// TIA Portal V17 export
// export: Created 2025-06-26T06:49:19.2186578Z, ExportSetting WithDefaults, DisplayName Totally Integrated Automation Portal, DisplayVersion V17 Update 8, DisplayName TIA Portal Openness, DisplayVersion V17 Update 8, DisplayName TIA Portal Version Control Interface, DisplayVersion V17, DisplayName STEP 7 Professional, DisplayVersion V17 Update 8, DisplayName STEP 7 Safety, DisplayVersion V17 Update 6, DisplayName WinCC Advanced, DisplayVersion V17 Update 8
FUNCTION "WinCCAlarmHandling" : Void   // FC24, FBD
TITLE = Convert alarms to WinCC format
{ S7_Optimized_Access := 'TRUE' }
VERSION : 0.1
// stored: AutoNumber true, IsIECCheckEnabled false, SetENOAutomatically false, UDAEnableTagReadback false
BEGIN

REGION Network 1 (SCL): Comments
   (*
   For every alarm that should appear in the HMI, it has to be translated into WinCC's alarm format
   This is a very "dumb" way to do it, but the advantage is it's easy to understand and easy to modify.

   Steps to add a new alarm:
   1. Add an entry in DB_WinCCAlarms under the right category
   2. Add a network in this FC with a WinCCAlarm block
   3. In the WinCC project, import the tag from DB_WinCCAlarms
   4. In the WinCC project, create an alarm which references this tag
   *)
END_REGION

REGION Network 2: 0001
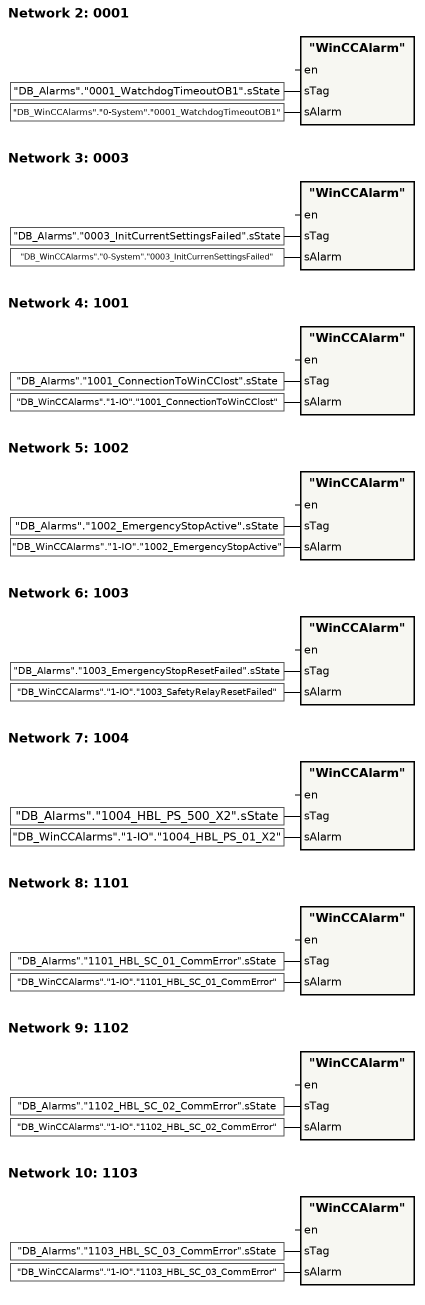
   "WinCCAlarm"(sTag := "DB_Alarms"."0001_WatchdogTimeoutOB1".sState,
                sAlarm := "DB_WinCCAlarms"."0-System"."0001_WatchdogTimeoutOB1");
END_REGION

REGION Network 3: 0003
   "WinCCAlarm"(sTag := "DB_Alarms"."0003_InitCurrentSettingsFailed".sState,
                sAlarm := "DB_WinCCAlarms"."0-System"."0003_InitCurrenSettingsFailed");
END_REGION

REGION Network 4: 1001
   "WinCCAlarm"(sTag := "DB_Alarms"."1001_ConnectionToWinCClost".sState,
                sAlarm := "DB_WinCCAlarms"."1-IO"."1001_ConnectionToWinCClost");
END_REGION

REGION Network 5: 1002
   "WinCCAlarm"(sTag := "DB_Alarms"."1002_EmergencyStopActive".sState,
                sAlarm := "DB_WinCCAlarms"."1-IO"."1002_EmergencyStopActive");
END_REGION

REGION Network 6: 1003
   "WinCCAlarm"(sTag := "DB_Alarms"."1003_EmergencyStopResetFailed".sState,
                sAlarm := "DB_WinCCAlarms"."1-IO"."1003_SafetyRelayResetFailed");
END_REGION

REGION Network 7: 1004
   "WinCCAlarm"(sTag := "DB_Alarms"."1004_HBL_PS_500_X2".sState,
                sAlarm := "DB_WinCCAlarms"."1-IO"."1004_HBL_PS_01_X2");
END_REGION

REGION Network 8: 1101
   "WinCCAlarm"(sTag := "DB_Alarms"."1101_HBL_SC_01_CommError".sState,
                sAlarm := "DB_WinCCAlarms"."1-IO"."1101_HBL_SC_01_CommError");
END_REGION

REGION Network 9: 1102
   "WinCCAlarm"(sTag := "DB_Alarms"."1102_HBL_SC_02_CommError".sState,
                sAlarm := "DB_WinCCAlarms"."1-IO"."1102_HBL_SC_02_CommError");
END_REGION

REGION Network 10: 1103
   "WinCCAlarm"(sTag := "DB_Alarms"."1103_HBL_SC_03_CommError".sState,
                sAlarm := "DB_WinCCAlarms"."1-IO"."1103_HBL_SC_03_CommError");
END_REGION

REGION Network 11: 1110
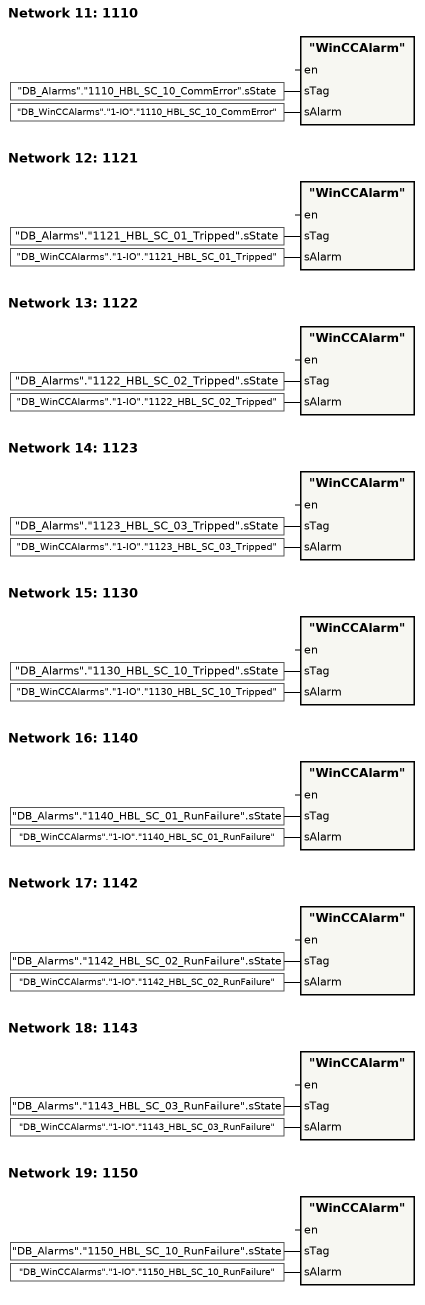
   "WinCCAlarm"(sTag := "DB_Alarms"."1110_HBL_SC_10_CommError".sState,
                sAlarm := "DB_WinCCAlarms"."1-IO"."1110_HBL_SC_10_CommError");
END_REGION

REGION Network 12: 1121
   "WinCCAlarm"(sTag := "DB_Alarms"."1121_HBL_SC_01_Tripped".sState,
                sAlarm := "DB_WinCCAlarms"."1-IO"."1121_HBL_SC_01_Tripped");
END_REGION

REGION Network 13: 1122
   "WinCCAlarm"(sTag := "DB_Alarms"."1122_HBL_SC_02_Tripped".sState,
                sAlarm := "DB_WinCCAlarms"."1-IO"."1122_HBL_SC_02_Tripped");
END_REGION

REGION Network 14: 1123
   "WinCCAlarm"(sTag := "DB_Alarms"."1123_HBL_SC_03_Tripped".sState,
                sAlarm := "DB_WinCCAlarms"."1-IO"."1123_HBL_SC_03_Tripped");
END_REGION

REGION Network 15: 1130
   "WinCCAlarm"(sTag := "DB_Alarms"."1130_HBL_SC_10_Tripped".sState,
                sAlarm := "DB_WinCCAlarms"."1-IO"."1130_HBL_SC_10_Tripped");
END_REGION

REGION Network 16: 1140
   "WinCCAlarm"(sTag := "DB_Alarms"."1140_HBL_SC_01_RunFailure".sState,
                sAlarm := "DB_WinCCAlarms"."1-IO"."1140_HBL_SC_01_RunFailure");
END_REGION

REGION Network 17: 1142
   "WinCCAlarm"(sTag := "DB_Alarms"."1142_HBL_SC_02_RunFailure".sState,
                sAlarm := "DB_WinCCAlarms"."1-IO"."1142_HBL_SC_02_RunFailure");
END_REGION

REGION Network 18: 1143
   "WinCCAlarm"(sTag := "DB_Alarms"."1143_HBL_SC_03_RunFailure".sState,
                sAlarm := "DB_WinCCAlarms"."1-IO"."1143_HBL_SC_03_RunFailure");
END_REGION

REGION Network 19: 1150
   "WinCCAlarm"(sTag := "DB_Alarms"."1150_HBL_SC_10_RunFailure".sState,
                sAlarm := "DB_WinCCAlarms"."1-IO"."1150_HBL_SC_10_RunFailure");
END_REGION

REGION Network 20: 1201
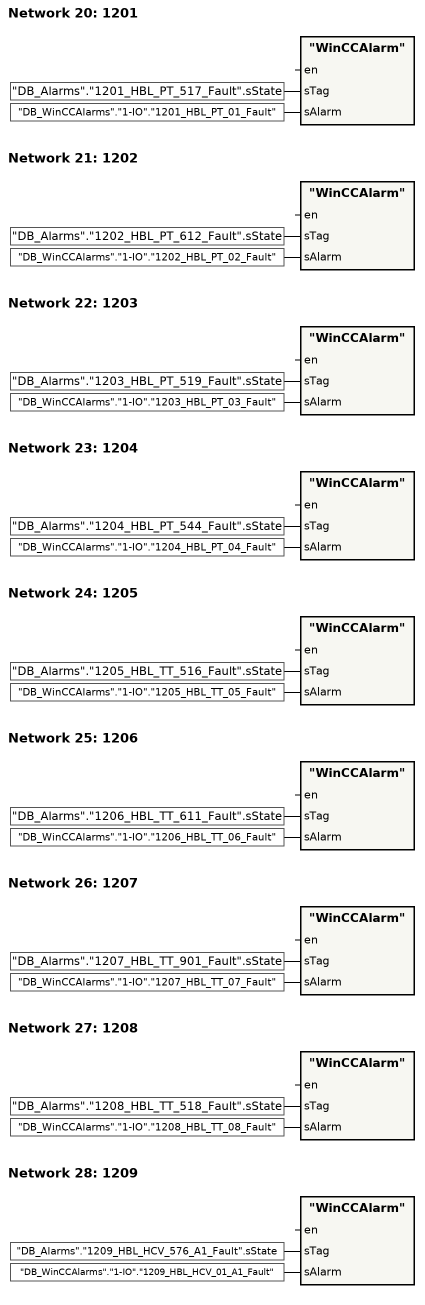
   "WinCCAlarm"(sTag := "DB_Alarms"."1201_HBL_PT_517_Fault".sState,
                sAlarm := "DB_WinCCAlarms"."1-IO"."1201_HBL_PT_01_Fault");
END_REGION

REGION Network 21: 1202
   "WinCCAlarm"(sTag := "DB_Alarms"."1202_HBL_PT_612_Fault".sState,
                sAlarm := "DB_WinCCAlarms"."1-IO"."1202_HBL_PT_02_Fault");
END_REGION

REGION Network 22: 1203
   "WinCCAlarm"(sTag := "DB_Alarms"."1203_HBL_PT_519_Fault".sState,
                sAlarm := "DB_WinCCAlarms"."1-IO"."1203_HBL_PT_03_Fault");
END_REGION

REGION Network 23: 1204
   "WinCCAlarm"(sTag := "DB_Alarms"."1204_HBL_PT_544_Fault".sState,
                sAlarm := "DB_WinCCAlarms"."1-IO"."1204_HBL_PT_04_Fault");
END_REGION

REGION Network 24: 1205
   "WinCCAlarm"(sTag := "DB_Alarms"."1205_HBL_TT_516_Fault".sState,
                sAlarm := "DB_WinCCAlarms"."1-IO"."1205_HBL_TT_05_Fault");
END_REGION

REGION Network 25: 1206
   "WinCCAlarm"(sTag := "DB_Alarms"."1206_HBL_TT_611_Fault".sState,
                sAlarm := "DB_WinCCAlarms"."1-IO"."1206_HBL_TT_06_Fault");
END_REGION

REGION Network 26: 1207
   "WinCCAlarm"(sTag := "DB_Alarms"."1207_HBL_TT_901_Fault".sState,
                sAlarm := "DB_WinCCAlarms"."1-IO"."1207_HBL_TT_07_Fault");
END_REGION

REGION Network 27: 1208
   "WinCCAlarm"(sTag := "DB_Alarms"."1208_HBL_TT_518_Fault".sState,
                sAlarm := "DB_WinCCAlarms"."1-IO"."1208_HBL_TT_08_Fault");
END_REGION

REGION Network 28: 1209
   "WinCCAlarm"(sTag := "DB_Alarms"."1209_HBL_HCV_576_A1_Fault".sState,
                sAlarm := "DB_WinCCAlarms"."1-IO"."1209_HBL_HCV_01_A1_Fault");
END_REGION

REGION Network 29: 1210
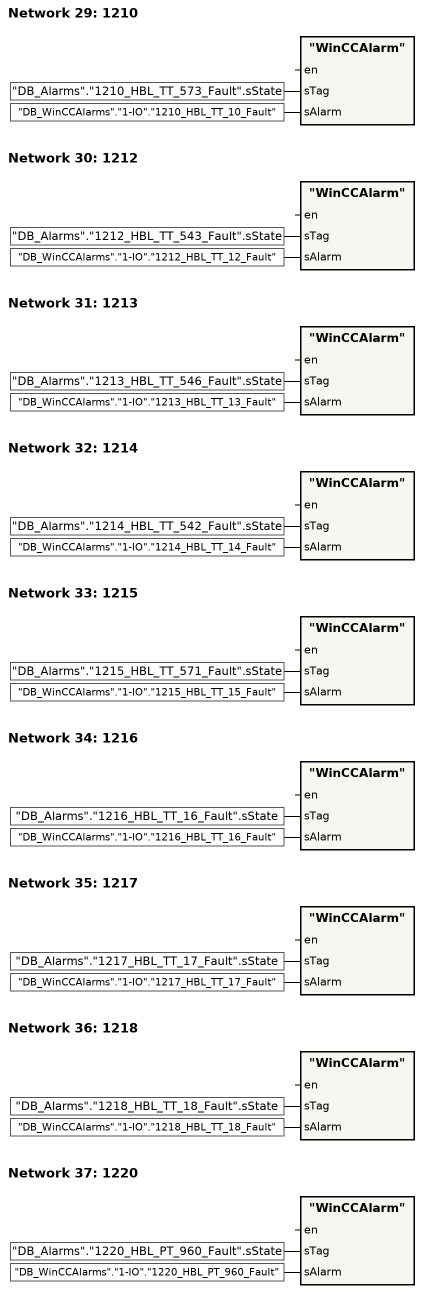
   "WinCCAlarm"(sTag := "DB_Alarms"."1210_HBL_TT_573_Fault".sState,
                sAlarm := "DB_WinCCAlarms"."1-IO"."1210_HBL_TT_10_Fault");
END_REGION

REGION Network 30: 1212
   "WinCCAlarm"(sTag := "DB_Alarms"."1212_HBL_TT_543_Fault".sState,
                sAlarm := "DB_WinCCAlarms"."1-IO"."1212_HBL_TT_12_Fault");
END_REGION

REGION Network 31: 1213
   "WinCCAlarm"(sTag := "DB_Alarms"."1213_HBL_TT_546_Fault".sState,
                sAlarm := "DB_WinCCAlarms"."1-IO"."1213_HBL_TT_13_Fault");
END_REGION

REGION Network 32: 1214
   "WinCCAlarm"(sTag := "DB_Alarms"."1214_HBL_TT_542_Fault".sState,
                sAlarm := "DB_WinCCAlarms"."1-IO"."1214_HBL_TT_14_Fault");
END_REGION

REGION Network 33: 1215
   "WinCCAlarm"(sTag := "DB_Alarms"."1215_HBL_TT_571_Fault".sState,
                sAlarm := "DB_WinCCAlarms"."1-IO"."1215_HBL_TT_15_Fault");
END_REGION

REGION Network 34: 1216
   "WinCCAlarm"(sTag := "DB_Alarms"."1216_HBL_TT_16_Fault".sState,
                sAlarm := "DB_WinCCAlarms"."1-IO"."1216_HBL_TT_16_Fault");
END_REGION

REGION Network 35: 1217
   "WinCCAlarm"(sTag := "DB_Alarms"."1217_HBL_TT_17_Fault".sState,
                sAlarm := "DB_WinCCAlarms"."1-IO"."1217_HBL_TT_17_Fault");
END_REGION

REGION Network 36: 1218
   "WinCCAlarm"(sTag := "DB_Alarms"."1218_HBL_TT_18_Fault".sState,
                sAlarm := "DB_WinCCAlarms"."1-IO"."1218_HBL_TT_18_Fault");
END_REGION

REGION Network 37: 1220
   "WinCCAlarm"(sTag := "DB_Alarms"."1220_HBL_PT_960_Fault".sState,
                sAlarm := "DB_WinCCAlarms"."1-IO"."1220_HBL_PT_960_Fault");
END_REGION

REGION Network 38: 1221
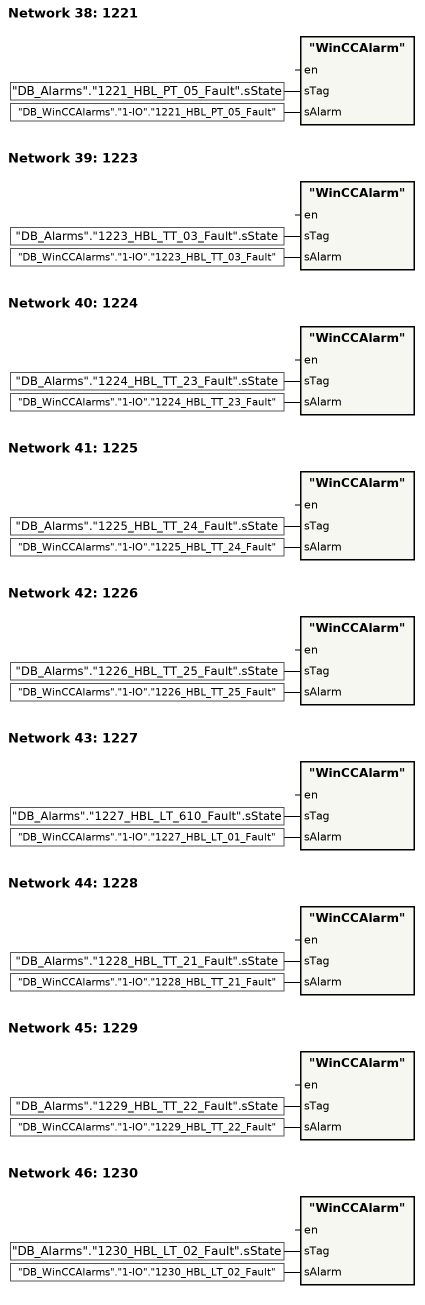
   "WinCCAlarm"(sTag := "DB_Alarms"."1221_HBL_PT_05_Fault".sState,
                sAlarm := "DB_WinCCAlarms"."1-IO"."1221_HBL_PT_05_Fault");
END_REGION

REGION Network 39: 1223
   "WinCCAlarm"(sTag := "DB_Alarms"."1223_HBL_TT_03_Fault".sState,
                sAlarm := "DB_WinCCAlarms"."1-IO"."1223_HBL_TT_03_Fault");
END_REGION

REGION Network 40: 1224
   "WinCCAlarm"(sTag := "DB_Alarms"."1224_HBL_TT_23_Fault".sState,
                sAlarm := "DB_WinCCAlarms"."1-IO"."1224_HBL_TT_23_Fault");
END_REGION

REGION Network 41: 1225
   "WinCCAlarm"(sTag := "DB_Alarms"."1225_HBL_TT_24_Fault".sState,
                sAlarm := "DB_WinCCAlarms"."1-IO"."1225_HBL_TT_24_Fault");
END_REGION

REGION Network 42: 1226
   "WinCCAlarm"(sTag := "DB_Alarms"."1226_HBL_TT_25_Fault".sState,
                sAlarm := "DB_WinCCAlarms"."1-IO"."1226_HBL_TT_25_Fault");
END_REGION

REGION Network 43: 1227
   "WinCCAlarm"(sTag := "DB_Alarms"."1227_HBL_LT_610_Fault".sState,
                sAlarm := "DB_WinCCAlarms"."1-IO"."1227_HBL_LT_01_Fault");
END_REGION

REGION Network 44: 1228
   "WinCCAlarm"(sTag := "DB_Alarms"."1228_HBL_TT_21_Fault".sState,
                sAlarm := "DB_WinCCAlarms"."1-IO"."1228_HBL_TT_21_Fault");
END_REGION

REGION Network 45: 1229
   "WinCCAlarm"(sTag := "DB_Alarms"."1229_HBL_TT_22_Fault".sState,
                sAlarm := "DB_WinCCAlarms"."1-IO"."1229_HBL_TT_22_Fault");
END_REGION

REGION Network 46: 1230
   "WinCCAlarm"(sTag := "DB_Alarms"."1230_HBL_LT_02_Fault".sState,
                sAlarm := "DB_WinCCAlarms"."1-IO"."1230_HBL_LT_02_Fault");
END_REGION

REGION Network 47: 1231
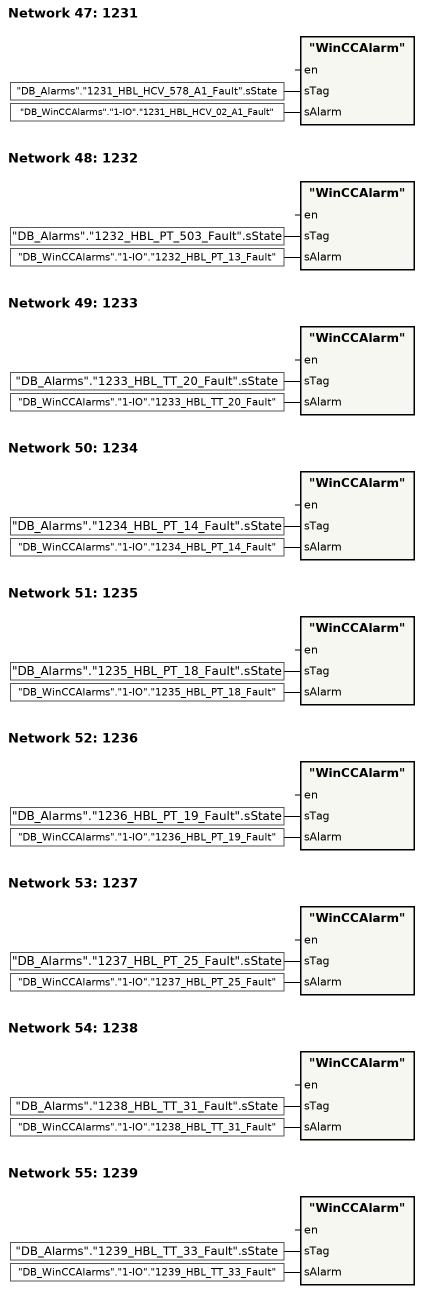
   "WinCCAlarm"(sTag := "DB_Alarms"."1231_HBL_HCV_578_A1_Fault".sState,
                sAlarm := "DB_WinCCAlarms"."1-IO"."1231_HBL_HCV_02_A1_Fault");
END_REGION

REGION Network 48: 1232
   "WinCCAlarm"(sTag := "DB_Alarms"."1232_HBL_PT_503_Fault".sState,
                sAlarm := "DB_WinCCAlarms"."1-IO"."1232_HBL_PT_13_Fault");
END_REGION

REGION Network 49: 1233
   "WinCCAlarm"(sTag := "DB_Alarms"."1233_HBL_TT_20_Fault".sState,
                sAlarm := "DB_WinCCAlarms"."1-IO"."1233_HBL_TT_20_Fault");
END_REGION

REGION Network 50: 1234
   "WinCCAlarm"(sTag := "DB_Alarms"."1234_HBL_PT_14_Fault".sState,
                sAlarm := "DB_WinCCAlarms"."1-IO"."1234_HBL_PT_14_Fault");
END_REGION

REGION Network 51: 1235
   "WinCCAlarm"(sTag := "DB_Alarms"."1235_HBL_PT_18_Fault".sState,
                sAlarm := "DB_WinCCAlarms"."1-IO"."1235_HBL_PT_18_Fault");
END_REGION

REGION Network 52: 1236
   "WinCCAlarm"(sTag := "DB_Alarms"."1236_HBL_PT_19_Fault".sState,
                sAlarm := "DB_WinCCAlarms"."1-IO"."1236_HBL_PT_19_Fault");
END_REGION

REGION Network 53: 1237
   "WinCCAlarm"(sTag := "DB_Alarms"."1237_HBL_PT_25_Fault".sState,
                sAlarm := "DB_WinCCAlarms"."1-IO"."1237_HBL_PT_25_Fault");
END_REGION

REGION Network 54: 1238
   "WinCCAlarm"(sTag := "DB_Alarms"."1238_HBL_TT_31_Fault".sState,
                sAlarm := "DB_WinCCAlarms"."1-IO"."1238_HBL_TT_31_Fault");
END_REGION

REGION Network 55: 1239
   "WinCCAlarm"(sTag := "DB_Alarms"."1239_HBL_TT_33_Fault".sState,
                sAlarm := "DB_WinCCAlarms"."1-IO"."1239_HBL_TT_33_Fault");
END_REGION

REGION Network 56: 1240
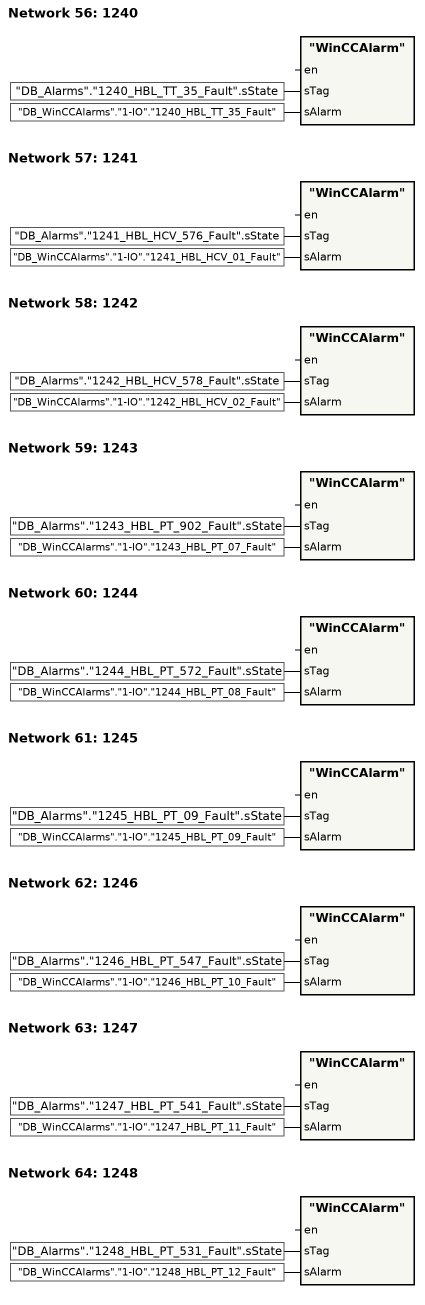
   "WinCCAlarm"(sTag := "DB_Alarms"."1240_HBL_TT_35_Fault".sState,
                sAlarm := "DB_WinCCAlarms"."1-IO"."1240_HBL_TT_35_Fault");
END_REGION

REGION Network 57: 1241
   "WinCCAlarm"(sTag := "DB_Alarms"."1241_HBL_HCV_576_Fault".sState,
                sAlarm := "DB_WinCCAlarms"."1-IO"."1241_HBL_HCV_01_Fault");
END_REGION

REGION Network 58: 1242
   "WinCCAlarm"(sTag := "DB_Alarms"."1242_HBL_HCV_578_Fault".sState,
                sAlarm := "DB_WinCCAlarms"."1-IO"."1242_HBL_HCV_02_Fault");
END_REGION

REGION Network 59: 1243
   "WinCCAlarm"(sTag := "DB_Alarms"."1243_HBL_PT_902_Fault".sState,
                sAlarm := "DB_WinCCAlarms"."1-IO"."1243_HBL_PT_07_Fault");
END_REGION

REGION Network 60: 1244
   "WinCCAlarm"(sTag := "DB_Alarms"."1244_HBL_PT_572_Fault".sState,
                sAlarm := "DB_WinCCAlarms"."1-IO"."1244_HBL_PT_08_Fault");
END_REGION

REGION Network 61: 1245
   "WinCCAlarm"(sTag := "DB_Alarms"."1245_HBL_PT_09_Fault".sState,
                sAlarm := "DB_WinCCAlarms"."1-IO"."1245_HBL_PT_09_Fault");
END_REGION

REGION Network 62: 1246
   "WinCCAlarm"(sTag := "DB_Alarms"."1246_HBL_PT_547_Fault".sState,
                sAlarm := "DB_WinCCAlarms"."1-IO"."1246_HBL_PT_10_Fault");
END_REGION

REGION Network 63: 1247
   "WinCCAlarm"(sTag := "DB_Alarms"."1247_HBL_PT_541_Fault".sState,
                sAlarm := "DB_WinCCAlarms"."1-IO"."1247_HBL_PT_11_Fault");
END_REGION

REGION Network 64: 1248
   "WinCCAlarm"(sTag := "DB_Alarms"."1248_HBL_PT_531_Fault".sState,
                sAlarm := "DB_WinCCAlarms"."1-IO"."1248_HBL_PT_12_Fault");
END_REGION

REGION Network 65: 1249
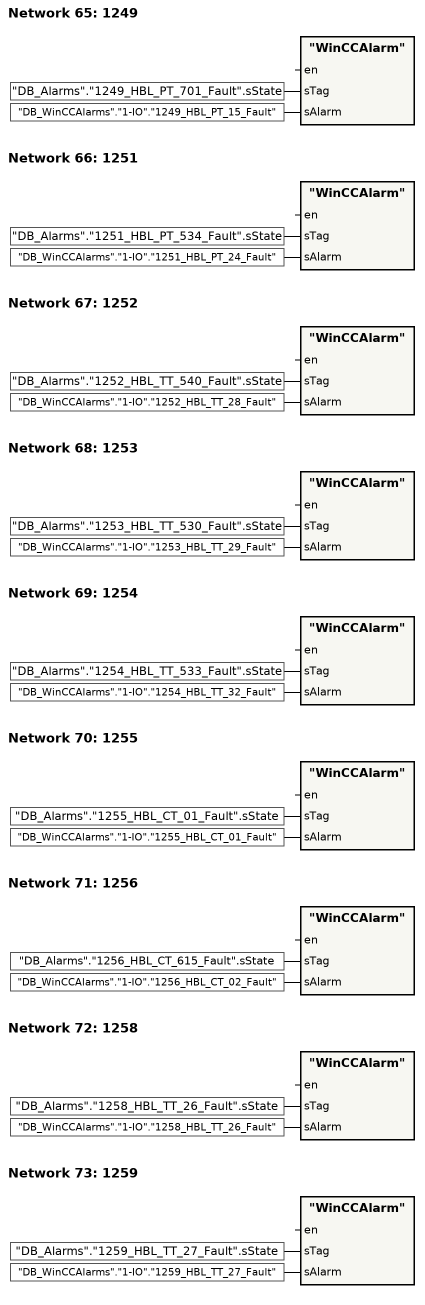
   "WinCCAlarm"(sTag := "DB_Alarms"."1249_HBL_PT_701_Fault".sState,
                sAlarm := "DB_WinCCAlarms"."1-IO"."1249_HBL_PT_15_Fault");
END_REGION

REGION Network 66: 1251
   "WinCCAlarm"(sTag := "DB_Alarms"."1251_HBL_PT_534_Fault".sState,
                sAlarm := "DB_WinCCAlarms"."1-IO"."1251_HBL_PT_24_Fault");
END_REGION

REGION Network 67: 1252
   "WinCCAlarm"(sTag := "DB_Alarms"."1252_HBL_TT_540_Fault".sState,
                sAlarm := "DB_WinCCAlarms"."1-IO"."1252_HBL_TT_28_Fault");
END_REGION

REGION Network 68: 1253
   "WinCCAlarm"(sTag := "DB_Alarms"."1253_HBL_TT_530_Fault".sState,
                sAlarm := "DB_WinCCAlarms"."1-IO"."1253_HBL_TT_29_Fault");
END_REGION

REGION Network 69: 1254
   "WinCCAlarm"(sTag := "DB_Alarms"."1254_HBL_TT_533_Fault".sState,
                sAlarm := "DB_WinCCAlarms"."1-IO"."1254_HBL_TT_32_Fault");
END_REGION

REGION Network 70: 1255
   "WinCCAlarm"(sTag := "DB_Alarms"."1255_HBL_CT_01_Fault".sState,
                sAlarm := "DB_WinCCAlarms"."1-IO"."1255_HBL_CT_01_Fault");
END_REGION

REGION Network 71: 1256
   "WinCCAlarm"(sTag := "DB_Alarms"."1256_HBL_CT_615_Fault".sState,
                sAlarm := "DB_WinCCAlarms"."1-IO"."1256_HBL_CT_02_Fault");
END_REGION

REGION Network 72: 1258
   "WinCCAlarm"(sTag := "DB_Alarms"."1258_HBL_TT_26_Fault".sState,
                sAlarm := "DB_WinCCAlarms"."1-IO"."1258_HBL_TT_26_Fault");
END_REGION

REGION Network 73: 1259
   "WinCCAlarm"(sTag := "DB_Alarms"."1259_HBL_TT_27_Fault".sState,
                sAlarm := "DB_WinCCAlarms"."1-IO"."1259_HBL_TT_27_Fault");
END_REGION

REGION Network 74: 1260
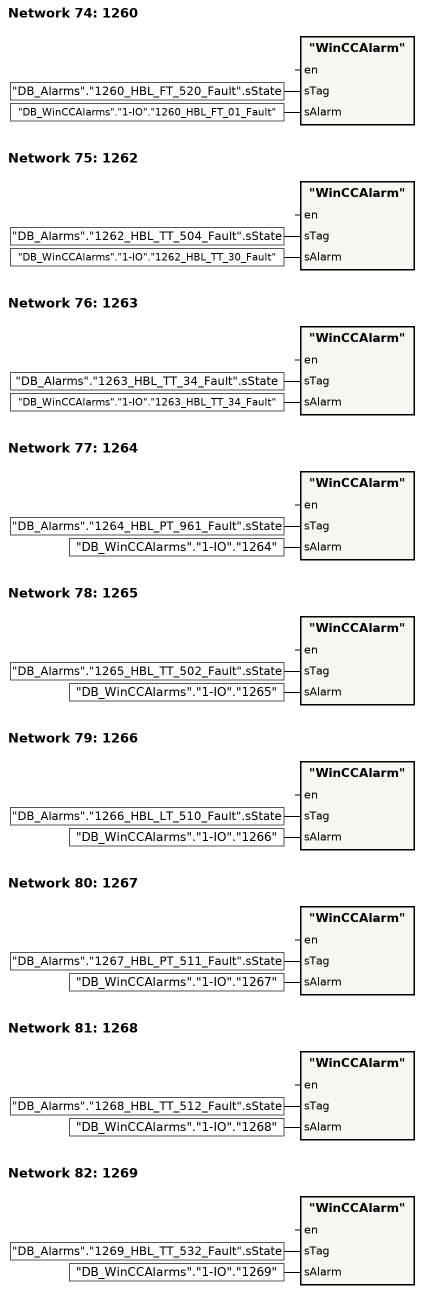
   "WinCCAlarm"(sTag := "DB_Alarms"."1260_HBL_FT_520_Fault".sState,
                sAlarm := "DB_WinCCAlarms"."1-IO"."1260_HBL_FT_01_Fault");
END_REGION

REGION Network 75: 1262
   "WinCCAlarm"(sTag := "DB_Alarms"."1262_HBL_TT_504_Fault".sState,
                sAlarm := "DB_WinCCAlarms"."1-IO"."1262_HBL_TT_30_Fault");
END_REGION

REGION Network 76: 1263
   "WinCCAlarm"(sTag := "DB_Alarms"."1263_HBL_TT_34_Fault".sState,
                sAlarm := "DB_WinCCAlarms"."1-IO"."1263_HBL_TT_34_Fault");
END_REGION

REGION Network 77: 1264
   "WinCCAlarm"(sTag := "DB_Alarms"."1264_HBL_PT_961_Fault".sState, sAlarm := "DB_WinCCAlarms"."1-IO"."1264");
END_REGION

REGION Network 78: 1265
   "WinCCAlarm"(sTag := "DB_Alarms"."1265_HBL_TT_502_Fault".sState, sAlarm := "DB_WinCCAlarms"."1-IO"."1265");
END_REGION

REGION Network 79: 1266
   "WinCCAlarm"(sTag := "DB_Alarms"."1266_HBL_LT_510_Fault".sState, sAlarm := "DB_WinCCAlarms"."1-IO"."1266");
END_REGION

REGION Network 80: 1267
   "WinCCAlarm"(sTag := "DB_Alarms"."1267_HBL_PT_511_Fault".sState, sAlarm := "DB_WinCCAlarms"."1-IO"."1267");
END_REGION

REGION Network 81: 1268
   "WinCCAlarm"(sTag := "DB_Alarms"."1268_HBL_TT_512_Fault".sState, sAlarm := "DB_WinCCAlarms"."1-IO"."1268");
END_REGION

REGION Network 82: 1269
   "WinCCAlarm"(sTag := "DB_Alarms"."1269_HBL_TT_532_Fault".sState, sAlarm := "DB_WinCCAlarms"."1-IO"."1269");
END_REGION

REGION Network 83: 1270
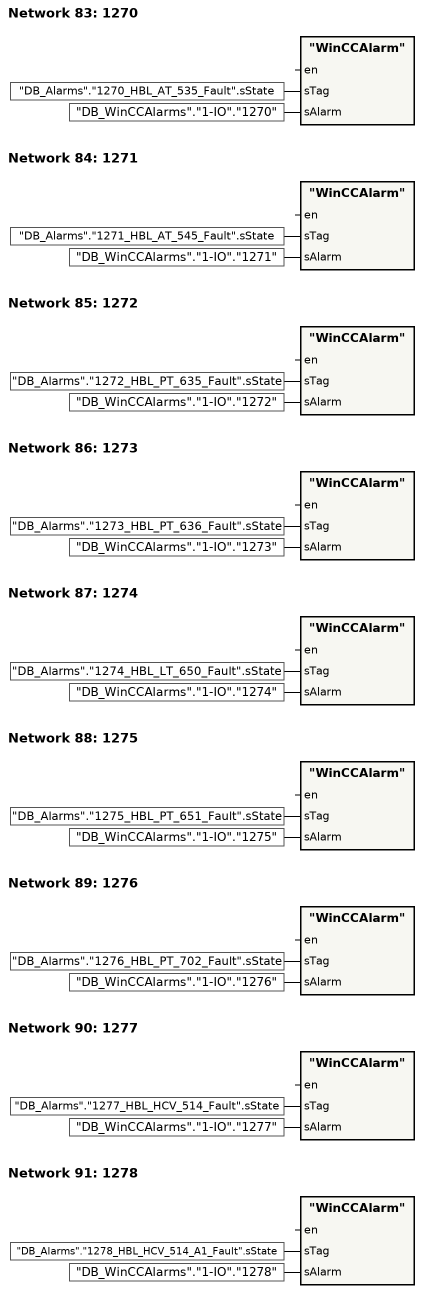
   "WinCCAlarm"(sTag := "DB_Alarms"."1270_HBL_AT_535_Fault".sState, sAlarm := "DB_WinCCAlarms"."1-IO"."1270");
END_REGION

REGION Network 84: 1271
   "WinCCAlarm"(sTag := "DB_Alarms"."1271_HBL_AT_545_Fault".sState, sAlarm := "DB_WinCCAlarms"."1-IO"."1271");
END_REGION

REGION Network 85: 1272
   "WinCCAlarm"(sTag := "DB_Alarms"."1272_HBL_PT_635_Fault".sState, sAlarm := "DB_WinCCAlarms"."1-IO"."1272");
END_REGION

REGION Network 86: 1273
   "WinCCAlarm"(sTag := "DB_Alarms"."1273_HBL_PT_636_Fault".sState, sAlarm := "DB_WinCCAlarms"."1-IO"."1273");
END_REGION

REGION Network 87: 1274
   "WinCCAlarm"(sTag := "DB_Alarms"."1274_HBL_LT_650_Fault".sState, sAlarm := "DB_WinCCAlarms"."1-IO"."1274");
END_REGION

REGION Network 88: 1275
   "WinCCAlarm"(sTag := "DB_Alarms"."1275_HBL_PT_651_Fault".sState, sAlarm := "DB_WinCCAlarms"."1-IO"."1275");
END_REGION

REGION Network 89: 1276
   "WinCCAlarm"(sTag := "DB_Alarms"."1276_HBL_PT_702_Fault".sState, sAlarm := "DB_WinCCAlarms"."1-IO"."1276");
END_REGION

REGION Network 90: 1277
   "WinCCAlarm"(sTag := "DB_Alarms"."1277_HBL_HCV_514_Fault".sState, sAlarm := "DB_WinCCAlarms"."1-IO"."1277");
END_REGION

REGION Network 91: 1278
   "WinCCAlarm"(sTag := "DB_Alarms"."1278_HBL_HCV_514_A1_Fault".sState,
                sAlarm := "DB_WinCCAlarms"."1-IO"."1278");
END_REGION

REGION Network 92: 1279
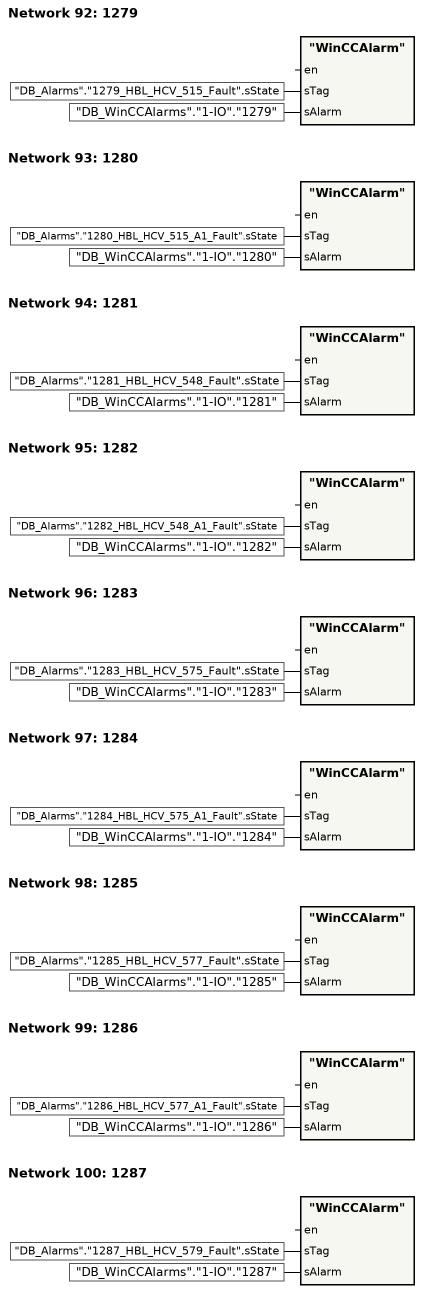
   "WinCCAlarm"(sTag := "DB_Alarms"."1279_HBL_HCV_515_Fault".sState, sAlarm := "DB_WinCCAlarms"."1-IO"."1279");
END_REGION

REGION Network 93: 1280
   "WinCCAlarm"(sTag := "DB_Alarms"."1280_HBL_HCV_515_A1_Fault".sState,
                sAlarm := "DB_WinCCAlarms"."1-IO"."1280");
END_REGION

REGION Network 94: 1281
   "WinCCAlarm"(sTag := "DB_Alarms"."1281_HBL_HCV_548_Fault".sState, sAlarm := "DB_WinCCAlarms"."1-IO"."1281");
END_REGION

REGION Network 95: 1282
   "WinCCAlarm"(sTag := "DB_Alarms"."1282_HBL_HCV_548_A1_Fault".sState,
                sAlarm := "DB_WinCCAlarms"."1-IO"."1282");
END_REGION

REGION Network 96: 1283
   "WinCCAlarm"(sTag := "DB_Alarms"."1283_HBL_HCV_575_Fault".sState, sAlarm := "DB_WinCCAlarms"."1-IO"."1283");
END_REGION

REGION Network 97: 1284
   "WinCCAlarm"(sTag := "DB_Alarms"."1284_HBL_HCV_575_A1_Fault".sState,
                sAlarm := "DB_WinCCAlarms"."1-IO"."1284");
END_REGION

REGION Network 98: 1285
   "WinCCAlarm"(sTag := "DB_Alarms"."1285_HBL_HCV_577_Fault".sState, sAlarm := "DB_WinCCAlarms"."1-IO"."1285");
END_REGION

REGION Network 99: 1286
   "WinCCAlarm"(sTag := "DB_Alarms"."1286_HBL_HCV_577_A1_Fault".sState,
                sAlarm := "DB_WinCCAlarms"."1-IO"."1286");
END_REGION

REGION Network 100: 1287
   "WinCCAlarm"(sTag := "DB_Alarms"."1287_HBL_HCV_579_Fault".sState, sAlarm := "DB_WinCCAlarms"."1-IO"."1287");
END_REGION

REGION Network 101: 1288
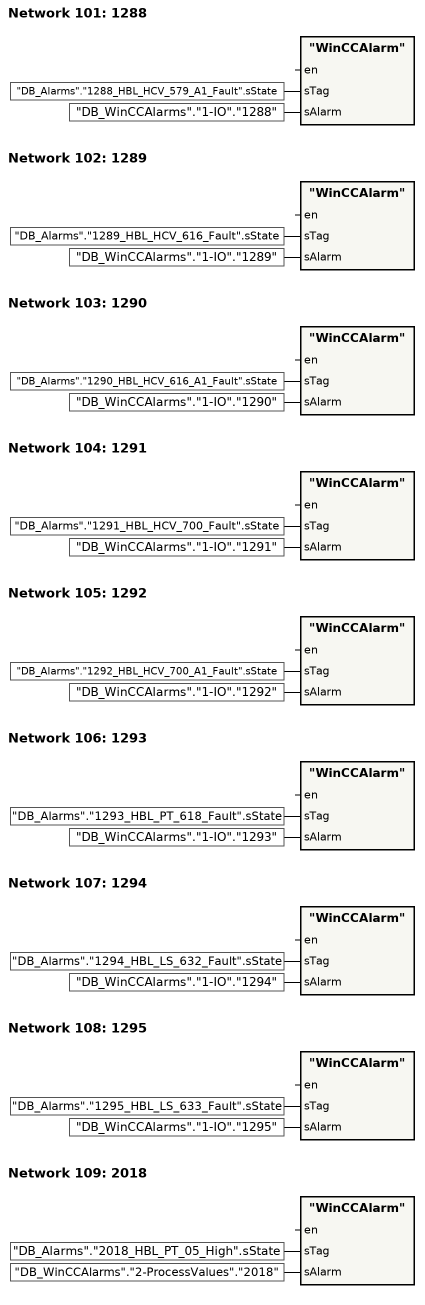
   "WinCCAlarm"(sTag := "DB_Alarms"."1288_HBL_HCV_579_A1_Fault".sState,
                sAlarm := "DB_WinCCAlarms"."1-IO"."1288");
END_REGION

REGION Network 102: 1289
   "WinCCAlarm"(sTag := "DB_Alarms"."1289_HBL_HCV_616_Fault".sState, sAlarm := "DB_WinCCAlarms"."1-IO"."1289");
END_REGION

REGION Network 103: 1290
   "WinCCAlarm"(sTag := "DB_Alarms"."1290_HBL_HCV_616_A1_Fault".sState,
                sAlarm := "DB_WinCCAlarms"."1-IO"."1290");
END_REGION

REGION Network 104: 1291
   "WinCCAlarm"(sTag := "DB_Alarms"."1291_HBL_HCV_700_Fault".sState, sAlarm := "DB_WinCCAlarms"."1-IO"."1291");
END_REGION

REGION Network 105: 1292
   "WinCCAlarm"(sTag := "DB_Alarms"."1292_HBL_HCV_700_A1_Fault".sState,
                sAlarm := "DB_WinCCAlarms"."1-IO"."1292");
END_REGION

REGION Network 106: 1293
   "WinCCAlarm"(sTag := "DB_Alarms"."1293_HBL_PT_618_Fault".sState, sAlarm := "DB_WinCCAlarms"."1-IO"."1293");
END_REGION

REGION Network 107: 1294
   "WinCCAlarm"(sTag := "DB_Alarms"."1294_HBL_LS_632_Fault".sState, sAlarm := "DB_WinCCAlarms"."1-IO"."1294");
END_REGION

REGION Network 108: 1295
   "WinCCAlarm"(sTag := "DB_Alarms"."1295_HBL_LS_633_Fault".sState, sAlarm := "DB_WinCCAlarms"."1-IO"."1295");
END_REGION

REGION Network 109: 2018
   "WinCCAlarm"(sTag := "DB_Alarms"."2018_HBL_PT_05_High".sState,
                sAlarm := "DB_WinCCAlarms"."2-ProcessValues"."2018");
END_REGION

REGION Network 110: 2028
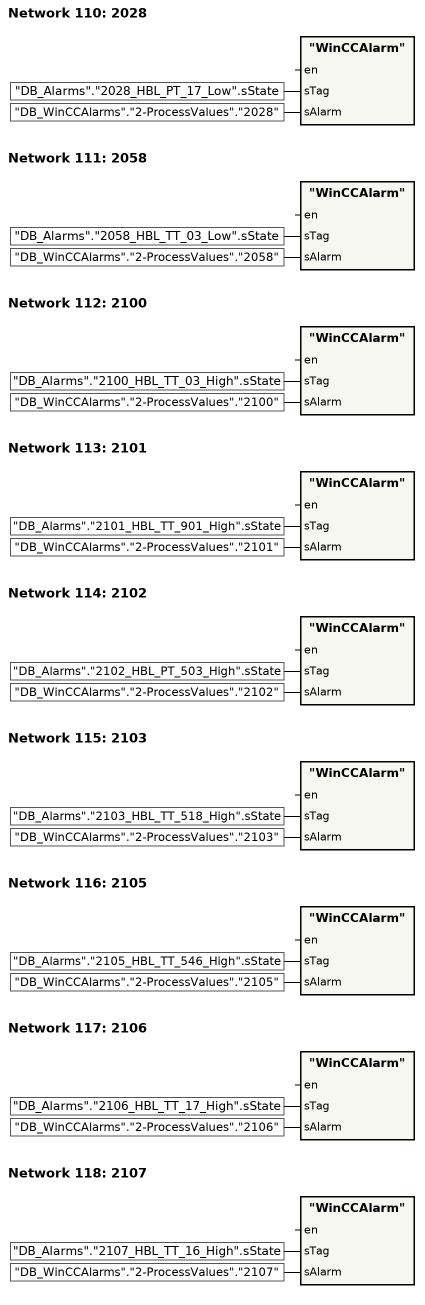
   "WinCCAlarm"(sTag := "DB_Alarms"."2028_HBL_PT_17_Low".sState,
                sAlarm := "DB_WinCCAlarms"."2-ProcessValues"."2028");
END_REGION

REGION Network 111: 2058
   "WinCCAlarm"(sTag := "DB_Alarms"."2058_HBL_TT_03_Low".sState,
                sAlarm := "DB_WinCCAlarms"."2-ProcessValues"."2058");
END_REGION

REGION Network 112: 2100
   "WinCCAlarm"(sTag := "DB_Alarms"."2100_HBL_TT_03_High".sState,
                sAlarm := "DB_WinCCAlarms"."2-ProcessValues"."2100");
END_REGION

REGION Network 113: 2101
   "WinCCAlarm"(sTag := "DB_Alarms"."2101_HBL_TT_901_High".sState,
                sAlarm := "DB_WinCCAlarms"."2-ProcessValues"."2101");
END_REGION

REGION Network 114: 2102
   "WinCCAlarm"(sTag := "DB_Alarms"."2102_HBL_PT_503_High".sState,
                sAlarm := "DB_WinCCAlarms"."2-ProcessValues"."2102");
END_REGION

REGION Network 115: 2103
   "WinCCAlarm"(sTag := "DB_Alarms"."2103_HBL_TT_518_High".sState,
                sAlarm := "DB_WinCCAlarms"."2-ProcessValues"."2103");
END_REGION

REGION Network 116: 2105
   "WinCCAlarm"(sTag := "DB_Alarms"."2105_HBL_TT_546_High".sState,
                sAlarm := "DB_WinCCAlarms"."2-ProcessValues"."2105");
END_REGION

REGION Network 117: 2106
   "WinCCAlarm"(sTag := "DB_Alarms"."2106_HBL_TT_17_High".sState,
                sAlarm := "DB_WinCCAlarms"."2-ProcessValues"."2106");
END_REGION

REGION Network 118: 2107
   "WinCCAlarm"(sTag := "DB_Alarms"."2107_HBL_TT_16_High".sState,
                sAlarm := "DB_WinCCAlarms"."2-ProcessValues"."2107");
END_REGION

REGION Network 119: 2108
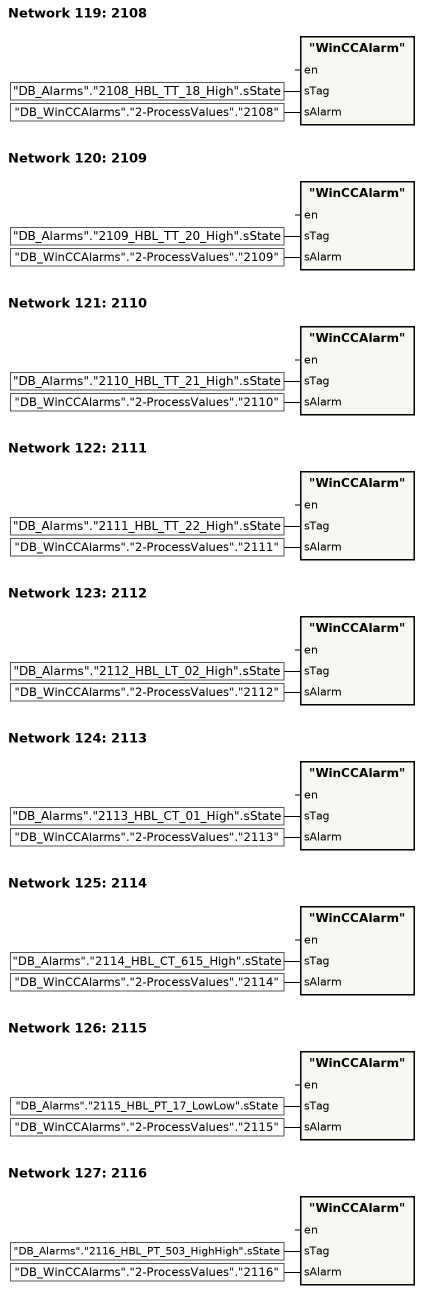
   "WinCCAlarm"(sTag := "DB_Alarms"."2108_HBL_TT_18_High".sState,
                sAlarm := "DB_WinCCAlarms"."2-ProcessValues"."2108");
END_REGION

REGION Network 120: 2109
   "WinCCAlarm"(sTag := "DB_Alarms"."2109_HBL_TT_20_High".sState,
                sAlarm := "DB_WinCCAlarms"."2-ProcessValues"."2109");
END_REGION

REGION Network 121: 2110
   "WinCCAlarm"(sTag := "DB_Alarms"."2110_HBL_TT_21_High".sState,
                sAlarm := "DB_WinCCAlarms"."2-ProcessValues"."2110");
END_REGION

REGION Network 122: 2111
   "WinCCAlarm"(sTag := "DB_Alarms"."2111_HBL_TT_22_High".sState,
                sAlarm := "DB_WinCCAlarms"."2-ProcessValues"."2111");
END_REGION

REGION Network 123: 2112
   "WinCCAlarm"(sTag := "DB_Alarms"."2112_HBL_LT_02_High".sState,
                sAlarm := "DB_WinCCAlarms"."2-ProcessValues"."2112");
END_REGION

REGION Network 124: 2113
   "WinCCAlarm"(sTag := "DB_Alarms"."2113_HBL_CT_01_High".sState,
                sAlarm := "DB_WinCCAlarms"."2-ProcessValues"."2113");
END_REGION

REGION Network 125: 2114
   "WinCCAlarm"(sTag := "DB_Alarms"."2114_HBL_CT_615_High".sState,
                sAlarm := "DB_WinCCAlarms"."2-ProcessValues"."2114");
END_REGION

REGION Network 126: 2115
   "WinCCAlarm"(sTag := "DB_Alarms"."2115_HBL_PT_17_LowLow".sState,
                sAlarm := "DB_WinCCAlarms"."2-ProcessValues"."2115");
END_REGION

REGION Network 127: 2116
   "WinCCAlarm"(sTag := "DB_Alarms"."2116_HBL_PT_503_HighHigh".sState,
                sAlarm := "DB_WinCCAlarms"."2-ProcessValues"."2116");
END_REGION

REGION Network 128: 2117
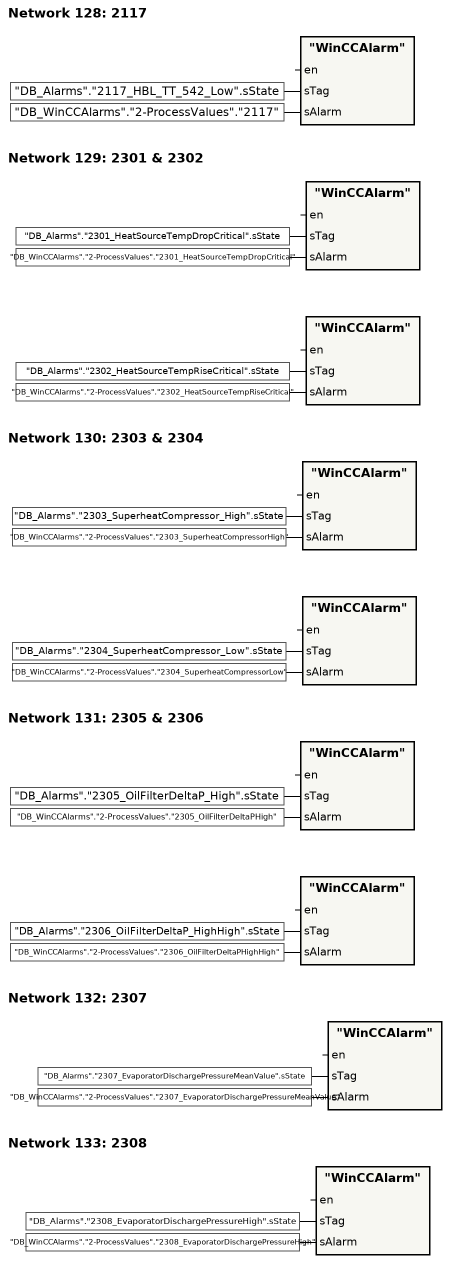
   "WinCCAlarm"(sTag := "DB_Alarms"."2117_HBL_TT_542_Low".sState,
                sAlarm := "DB_WinCCAlarms"."2-ProcessValues"."2117");
END_REGION

REGION Network 129: 2301 & 2302
   "WinCCAlarm"(sTag := "DB_Alarms"."2301_HeatSourceTempDropCritical".sState,
                sAlarm := "DB_WinCCAlarms"."2-ProcessValues"."2301_HeatSourceTempDropCritical");
   "WinCCAlarm"(sTag := "DB_Alarms"."2302_HeatSourceTempRiseCritical".sState,
                sAlarm := "DB_WinCCAlarms"."2-ProcessValues"."2302_HeatSourceTempRiseCritical");
END_REGION

REGION Network 130: 2303 & 2304
   "WinCCAlarm"(sTag := "DB_Alarms"."2303_SuperheatCompressor_High".sState,
                sAlarm := "DB_WinCCAlarms"."2-ProcessValues"."2303_SuperheatCompressorHigh");
   "WinCCAlarm"(sTag := "DB_Alarms"."2304_SuperheatCompressor_Low".sState,
                sAlarm := "DB_WinCCAlarms"."2-ProcessValues"."2304_SuperheatCompressorLow");
END_REGION

REGION Network 131: 2305 & 2306
   "WinCCAlarm"(sTag := "DB_Alarms"."2305_OilFilterDeltaP_High".sState,
                sAlarm := "DB_WinCCAlarms"."2-ProcessValues"."2305_OilFilterDeltaPHigh");
   "WinCCAlarm"(sTag := "DB_Alarms"."2306_OilFilterDeltaP_HighHigh".sState,
                sAlarm := "DB_WinCCAlarms"."2-ProcessValues"."2306_OilFilterDeltaPHighHigh");
END_REGION

REGION Network 132: 2307
   "WinCCAlarm"(sTag := "DB_Alarms"."2307_EvaporatorDischargePressureMeanValue".sState,
                sAlarm := "DB_WinCCAlarms"."2-ProcessValues"."2307_EvaporatorDischargePressureMeanValue");
END_REGION

REGION Network 133: 2308
   "WinCCAlarm"(sTag := "DB_Alarms"."2308_EvaporatorDischargePressureHigh".sState,
                sAlarm := "DB_WinCCAlarms"."2-ProcessValues"."2308_EvaporatorDischargePressureHigh");
END_REGION

REGION Network 134: 2309
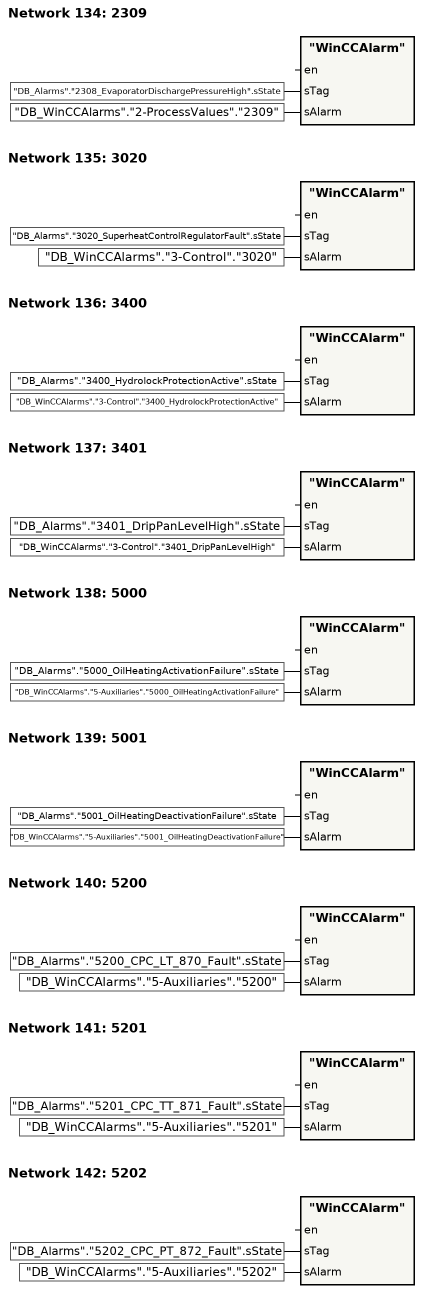
   "WinCCAlarm"(sTag := "DB_Alarms"."2308_EvaporatorDischargePressureHigh".sState,
                sAlarm := "DB_WinCCAlarms"."2-ProcessValues"."2309");
END_REGION

REGION Network 135: 3020
   "WinCCAlarm"(sTag := "DB_Alarms"."3020_SuperheatControlRegulatorFault".sState,
                sAlarm := "DB_WinCCAlarms"."3-Control"."3020");
END_REGION

REGION Network 136: 3400
   "WinCCAlarm"(sTag := "DB_Alarms"."3400_HydrolockProtectionActive".sState,
                sAlarm := "DB_WinCCAlarms"."3-Control"."3400_HydrolockProtectionActive");
END_REGION

REGION Network 137: 3401
   "WinCCAlarm"(sTag := "DB_Alarms"."3401_DripPanLevelHigh".sState,
                sAlarm := "DB_WinCCAlarms"."3-Control"."3401_DripPanLevelHigh");
END_REGION

REGION Network 138: 5000
   "WinCCAlarm"(sTag := "DB_Alarms"."5000_OilHeatingActivationFailure".sState,
                sAlarm := "DB_WinCCAlarms"."5-Auxiliaries"."5000_OilHeatingActivationFailure");
END_REGION

REGION Network 139: 5001
   "WinCCAlarm"(sTag := "DB_Alarms"."5001_OilHeatingDeactivationFailure".sState,
                sAlarm := "DB_WinCCAlarms"."5-Auxiliaries"."5001_OilHeatingDeactivationFailure");
END_REGION

REGION Network 140: 5200
   "WinCCAlarm"(sTag := "DB_Alarms"."5200_CPC_LT_870_Fault".sState,
                sAlarm := "DB_WinCCAlarms"."5-Auxiliaries"."5200");
END_REGION

REGION Network 141: 5201
   "WinCCAlarm"(sTag := "DB_Alarms"."5201_CPC_TT_871_Fault".sState,
                sAlarm := "DB_WinCCAlarms"."5-Auxiliaries"."5201");
END_REGION

REGION Network 142: 5202
   "WinCCAlarm"(sTag := "DB_Alarms"."5202_CPC_PT_872_Fault".sState,
                sAlarm := "DB_WinCCAlarms"."5-Auxiliaries"."5202");
END_REGION

REGION Network 143: 5203
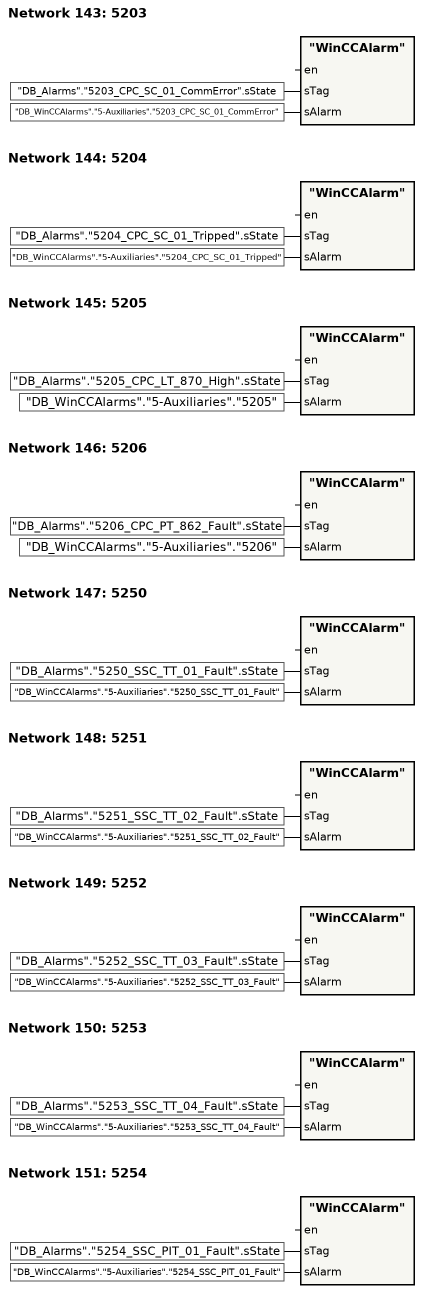
   "WinCCAlarm"(sTag := "DB_Alarms"."5203_CPC_SC_01_CommError".sState,
                sAlarm := "DB_WinCCAlarms"."5-Auxiliaries"."5203_CPC_SC_01_CommError");
END_REGION

REGION Network 144: 5204
   "WinCCAlarm"(sTag := "DB_Alarms"."5204_CPC_SC_01_Tripped".sState,
                sAlarm := "DB_WinCCAlarms"."5-Auxiliaries"."5204_CPC_SC_01_Tripped");
END_REGION

REGION Network 145: 5205
   "WinCCAlarm"(sTag := "DB_Alarms"."5205_CPC_LT_870_High".sState,
                sAlarm := "DB_WinCCAlarms"."5-Auxiliaries"."5205");
END_REGION

REGION Network 146: 5206
   "WinCCAlarm"(sTag := "DB_Alarms"."5206_CPC_PT_862_Fault".sState,
                sAlarm := "DB_WinCCAlarms"."5-Auxiliaries"."5206");
END_REGION

REGION Network 147: 5250
   "WinCCAlarm"(sTag := "DB_Alarms"."5250_SSC_TT_01_Fault".sState,
                sAlarm := "DB_WinCCAlarms"."5-Auxiliaries"."5250_SSC_TT_01_Fault");
END_REGION

REGION Network 148: 5251
   "WinCCAlarm"(sTag := "DB_Alarms"."5251_SSC_TT_02_Fault".sState,
                sAlarm := "DB_WinCCAlarms"."5-Auxiliaries"."5251_SSC_TT_02_Fault");
END_REGION

REGION Network 149: 5252
   "WinCCAlarm"(sTag := "DB_Alarms"."5252_SSC_TT_03_Fault".sState,
                sAlarm := "DB_WinCCAlarms"."5-Auxiliaries"."5252_SSC_TT_03_Fault");
END_REGION

REGION Network 150: 5253
   "WinCCAlarm"(sTag := "DB_Alarms"."5253_SSC_TT_04_Fault".sState,
                sAlarm := "DB_WinCCAlarms"."5-Auxiliaries"."5253_SSC_TT_04_Fault");
END_REGION

REGION Network 151: 5254
   "WinCCAlarm"(sTag := "DB_Alarms"."5254_SSC_PIT_01_Fault".sState,
                sAlarm := "DB_WinCCAlarms"."5-Auxiliaries"."5254_SSC_PIT_01_Fault");
END_REGION

REGION Network 152: 5255
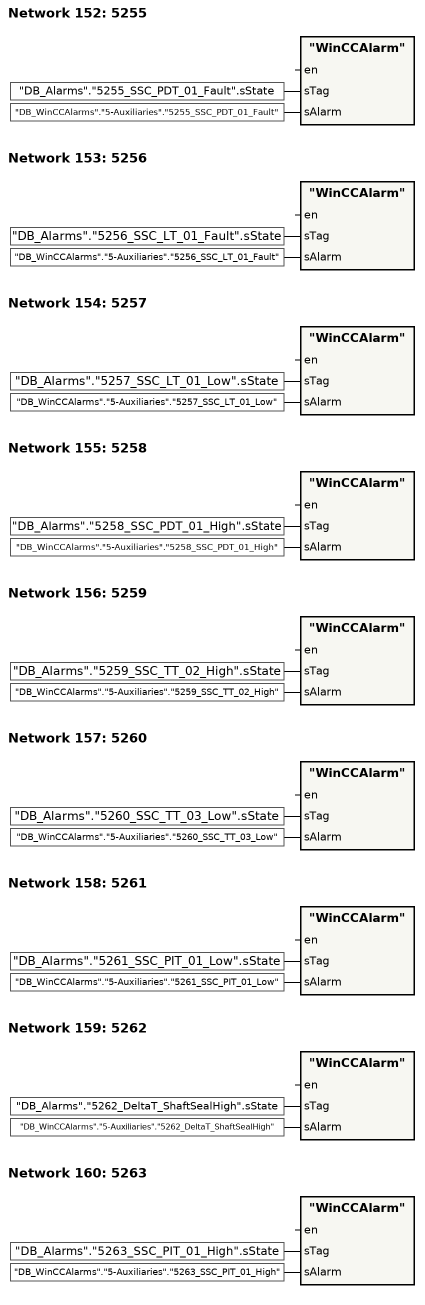
   "WinCCAlarm"(sTag := "DB_Alarms"."5255_SSC_PDT_01_Fault".sState,
                sAlarm := "DB_WinCCAlarms"."5-Auxiliaries"."5255_SSC_PDT_01_Fault");
END_REGION

REGION Network 153: 5256
   "WinCCAlarm"(sTag := "DB_Alarms"."5256_SSC_LT_01_Fault".sState,
                sAlarm := "DB_WinCCAlarms"."5-Auxiliaries"."5256_SSC_LT_01_Fault");
END_REGION

REGION Network 154: 5257
   "WinCCAlarm"(sTag := "DB_Alarms"."5257_SSC_LT_01_Low".sState,
                sAlarm := "DB_WinCCAlarms"."5-Auxiliaries"."5257_SSC_LT_01_Low");
END_REGION

REGION Network 155: 5258
   "WinCCAlarm"(sTag := "DB_Alarms"."5258_SSC_PDT_01_High".sState,
                sAlarm := "DB_WinCCAlarms"."5-Auxiliaries"."5258_SSC_PDT_01_High");
END_REGION

REGION Network 156: 5259
   "WinCCAlarm"(sTag := "DB_Alarms"."5259_SSC_TT_02_High".sState,
                sAlarm := "DB_WinCCAlarms"."5-Auxiliaries"."5259_SSC_TT_02_High");
END_REGION

REGION Network 157: 5260
   "WinCCAlarm"(sTag := "DB_Alarms"."5260_SSC_TT_03_Low".sState,
                sAlarm := "DB_WinCCAlarms"."5-Auxiliaries"."5260_SSC_TT_03_Low");
END_REGION

REGION Network 158: 5261
   "WinCCAlarm"(sTag := "DB_Alarms"."5261_SSC_PIT_01_Low".sState,
                sAlarm := "DB_WinCCAlarms"."5-Auxiliaries"."5261_SSC_PIT_01_Low");
END_REGION

REGION Network 159: 5262
   "WinCCAlarm"(sTag := "DB_Alarms"."5262_DeltaT_ShaftSealHigh".sState,
                sAlarm := "DB_WinCCAlarms"."5-Auxiliaries"."5262_DeltaT_ShaftSealHigh");
END_REGION

REGION Network 160: 5263
   "WinCCAlarm"(sTag := "DB_Alarms"."5263_SSC_PIT_01_High".sState,
                sAlarm := "DB_WinCCAlarms"."5-Auxiliaries"."5263_SSC_PIT_01_High");
END_REGION

REGION Network 161: 5268
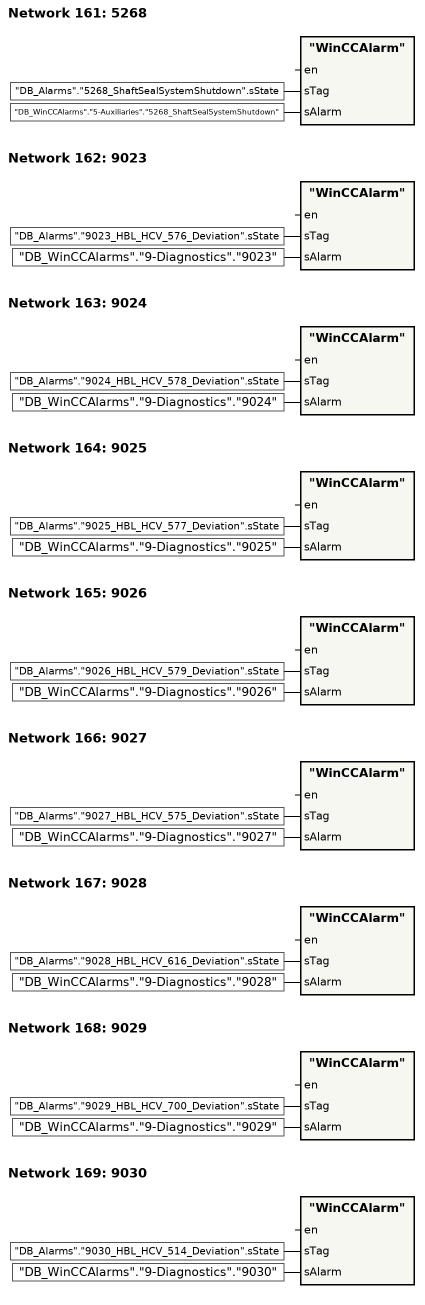
   "WinCCAlarm"(sTag := "DB_Alarms"."5268_ShaftSealSystemShutdown".sState,
                sAlarm := "DB_WinCCAlarms"."5-Auxiliaries"."5268_ShaftSealSystemShutdown");
END_REGION

REGION Network 162: 9023
   "WinCCAlarm"(sTag := "DB_Alarms"."9023_HBL_HCV_576_Deviation".sState,
                sAlarm := "DB_WinCCAlarms"."9-Diagnostics"."9023");
END_REGION

REGION Network 163: 9024
   "WinCCAlarm"(sTag := "DB_Alarms"."9024_HBL_HCV_578_Deviation".sState,
                sAlarm := "DB_WinCCAlarms"."9-Diagnostics"."9024");
END_REGION

REGION Network 164: 9025
   "WinCCAlarm"(sTag := "DB_Alarms"."9025_HBL_HCV_577_Deviation".sState,
                sAlarm := "DB_WinCCAlarms"."9-Diagnostics"."9025");
END_REGION

REGION Network 165: 9026
   "WinCCAlarm"(sTag := "DB_Alarms"."9026_HBL_HCV_579_Deviation".sState,
                sAlarm := "DB_WinCCAlarms"."9-Diagnostics"."9026");
END_REGION

REGION Network 166: 9027
   "WinCCAlarm"(sTag := "DB_Alarms"."9027_HBL_HCV_575_Deviation".sState,
                sAlarm := "DB_WinCCAlarms"."9-Diagnostics"."9027");
END_REGION

REGION Network 167: 9028
   "WinCCAlarm"(sTag := "DB_Alarms"."9028_HBL_HCV_616_Deviation".sState,
                sAlarm := "DB_WinCCAlarms"."9-Diagnostics"."9028");
END_REGION

REGION Network 168: 9029
   "WinCCAlarm"(sTag := "DB_Alarms"."9029_HBL_HCV_700_Deviation".sState,
                sAlarm := "DB_WinCCAlarms"."9-Diagnostics"."9029");
END_REGION

REGION Network 169: 9030
   "WinCCAlarm"(sTag := "DB_Alarms"."9030_HBL_HCV_514_Deviation".sState,
                sAlarm := "DB_WinCCAlarms"."9-Diagnostics"."9030");
END_REGION

REGION Network 170: 9031
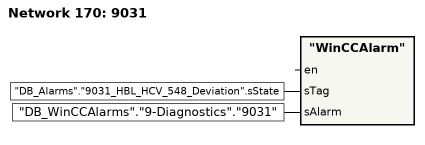
   "WinCCAlarm"(sTag := "DB_Alarms"."9031_HBL_HCV_548_Deviation".sState,
                sAlarm := "DB_WinCCAlarms"."9-Diagnostics"."9031");
END_REGION
END_FUNCTION
